% RSLogix 500 project digital filling station.RSS, saved by version 8.40.00.08 %
PROJECT "UNTITLED"    % processor: Bul.1763 MicroLogix 1100 Series B %

PROGRAM FILES
  LAD 2   3 rungs
  LAD 3 "IO"  8 rungs
  LAD 4 "CONTROLS"  4 rungs

DATA FILES
  O0 OUTPUT  4 elements
  I1 INPUT  6 elements
  S2 STATUS  66 elements
  B3 BINARY  1 elements
  T4 TIMER  1 elements
  C5 COUNTER  1 elements
  R6 CONTROL  1 elements
  N7 INTEGER  1 elements
  F8 FLOAT  1 elements

LADDER 2
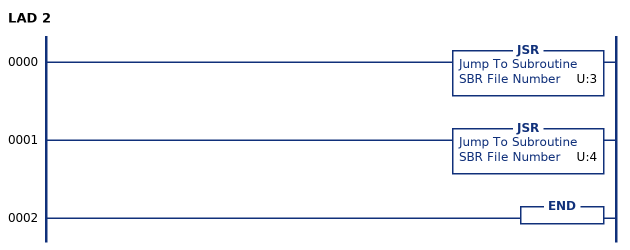
% Rung: 0 %
SOR JSR U:3 EOR
% Rung: 1 %
SOR JSR U:4 EOR
% Rung: 2 %
SOR END EOR

LADDER 3 "IO"
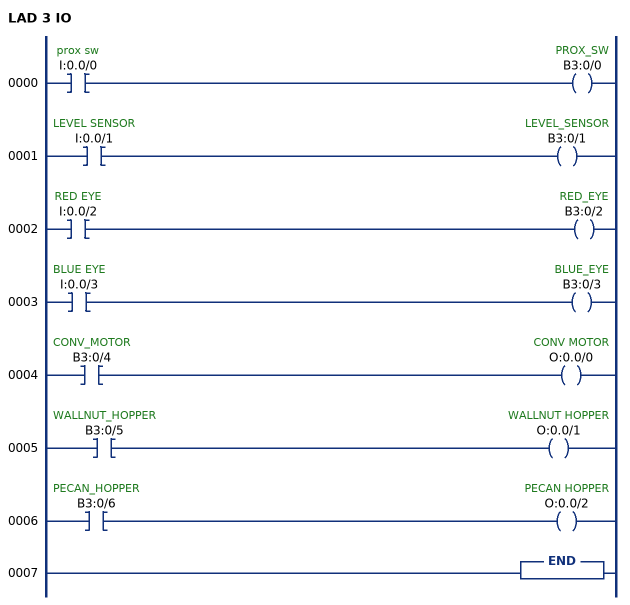
% Rung: 0 %
SOR XIC I:0.0/0 OTE B3:0/0 EOR
%   I:0.0/0  "prox sw" %
%   B3:0/0  PROX_SW %
% Rung: 1 %
SOR XIC I:0.0/1 OTE B3:0/1 EOR
%   I:0.0/1  "LEVEL SENSOR" %
%   B3:0/1  LEVEL_SENSOR %
% Rung: 2 %
SOR XIC I:0.0/2 OTE B3:0/2 EOR
%   I:0.0/2  "RED EYE" %
%   B3:0/2  RED_EYE %
% Rung: 3 %
SOR XIC I:0.0/3 OTE B3:0/3 EOR
%   I:0.0/3  "BLUE EYE" %
%   B3:0/3  BLUE_EYE %
% Rung: 4 %
SOR XIC B3:0/4 OTE O:0.0/0 EOR
%   B3:0/4  CONV_MOTOR %
%   O:0.0/0  "CONV MOTOR" %
% Rung: 5 %
SOR XIC B3:0/5 OTE O:0.0/1 EOR
%   B3:0/5  WALLNUT_HOPPER %
%   O:0.0/1  "WALLNUT HOPPER" %
% Rung: 6 %
SOR XIC B3:0/6 OTE O:0.0/2 EOR
%   B3:0/6  PECAN_HOPPER %
%   O:0.0/2  "PECAN HOPPER" %
% Rung: 7 %
SOR END EOR

LADDER 4 "CONTROLS"
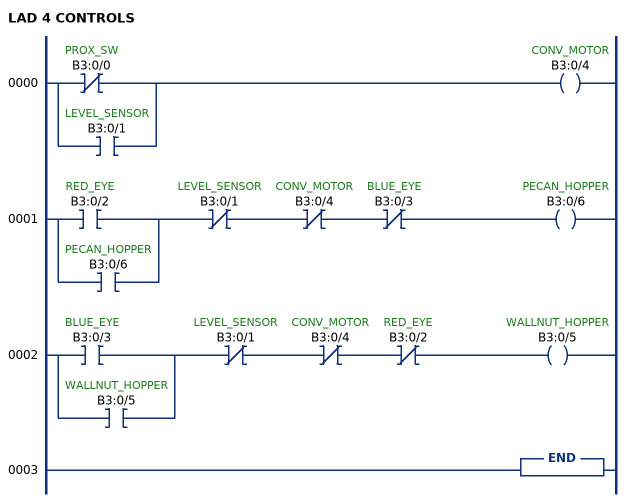
% Rung: 0 %
SOR BST XIO B3:0/0 NXB XIC B3:0/1 BND OTE B3:0/4 EOR
%   B3:0/0  PROX_SW %
%   B3:0/1  LEVEL_SENSOR %
%   B3:0/4  CONV_MOTOR %
% Rung: 1 %
SOR BST XIC B3:0/2 NXB XIC B3:0/6 BND XIO B3:0/1 XIO B3:0/4 XIO B3:0/3 OTE B3:0/6 EOR
%   B3:0/2  RED_EYE %
%   B3:0/6  PECAN_HOPPER %
%   B3:0/1  LEVEL_SENSOR %
%   B3:0/4  CONV_MOTOR %
%   B3:0/3  BLUE_EYE %
% Rung: 2 %
SOR BST XIC B3:0/3 NXB XIC B3:0/5 BND XIO B3:0/1 XIO B3:0/4 XIO B3:0/2 OTE B3:0/5 EOR
%   B3:0/3  BLUE_EYE %
%   B3:0/5  WALLNUT_HOPPER %
%   B3:0/1  LEVEL_SENSOR %
%   B3:0/4  CONV_MOTOR %
%   B3:0/2  RED_EYE %
% Rung: 3 %
SOR END EOR

DATA TABLE (non-zero values as saved)
DATA B3
% B3:0 % 0X001C
